{attribute 'GeneratedUsingTerminal: ER5101-0002-0019'}
{attribute addProperty BoxType "ER5101-0002-0019"}
{attribute addProperty Id "ENC_Status_compactAT %I*ENC_Status_compact_F4F8958316ENC_Control_compactAT %Q*ENC_Control_compact_E6DC9B254WcStateAT %I*WcState_9091E0EB2InfoDataAT %I*InfoData_94A18F5E2"}
{attribute addProperty CRC "56476779"}
{attribute addProperty Size "24"}
TYPE ER5101_035DC46B EXTENDS EtcSlaveTerminalBase_947E5A46 :
STRUCT
	{attribute addProperty Name "ENC_Status_compact"}
	ENC_Status_compact : ENC_Status_compact_F4F89583;
	{attribute addProperty Name "ENC_Control_compact"}
	ENC_Control_compact : ENC_Control_compact_E6DC9B25;
	{attribute addProperty Name "WcState"}
	WcState : WcState_9091E0EB;
	{attribute addProperty Name "InfoData"}
	InfoData : InfoData_94A18F5E;
END_STRUCT
END_TYPE

(* stored: Version 1.2.0.0, ProductVersion 3.1.4024.9
   DUT ER5101_035DC46B: Id {c64e6964-e6de-4bca-af83-979a42e15b39} *)
